{attribute addProperty BoxType "EK1122-0000-0018"}
{attribute addProperty Id "Beckhoff_APS4xxxsub_EK1100EK1100_179A0949162A_0001_APS4322_7000_0017APS4322_1E964C4E2242280.25"}
{attribute addProperty CRC "1708001423"}
{attribute addProperty SizeInBites "2258"}
{attribute addProperty SizeInBytes "282.25"}
TYPE Beckhoff_APS4xxxEK1122_65CE088F EXTENDS EK1122_179A0949 :
STRUCT
	{attribute addProperty Name "Beckhoff_APS4xxxsub_EK1100"}
	Beckhoff_APS4xxxsub_EK1100 : EK1100_179A0949;
	{attribute addProperty Name "A_0001_APS4322_7000_0017"}
	A_0001_APS4322_7000_0017 : APS4322_1E964C4E;
END_STRUCT
END_TYPE

(* stored: Version 1.2.0.0, ProductVersion 3.1.4024.9
   DUT Beckhoff_APS4xxxEK1122_65CE088F: Id {feda9cb7-3c17-47cb-a39d-0dc4819793db} *)
